{attribute 'qualified_only'}
VAR_GLOBAL
	station:typeStation; //data relating to the entire station
END_VAR

(* stored: Version 1.1.0.1, ProductVersion 3.1.4024.12
   GVL S6_Global: Id {0c991f4d-64f1-4dda-9163-b40c275a421c} *)
